(* PLC project Unnamed, Unknown Unnamed 1 *)
(* stored: creationDateTime 2012-09-12T23:30:19, modificationDateTime 2026-03-14T22:28:08 *)

FUNCTION_BLOCK getpybool
  VAR
    getpy : python_gear;
    latch : SR;
  END_VAR
  VAR_INPUT
    name : STRING;
  END_VAR
  VAR_OUTPUT
    val : BOOL;
  END_VAR
  VAR  (* added by the conversion: wires and edge detectors of the diagram *)
    _EQ41_ENO : BOOL;
    _EQ41_OUT : BOOL;
    _EQ3_ENO : BOOL;
    _EQ3_OUT : BOOL;
  END_VAR

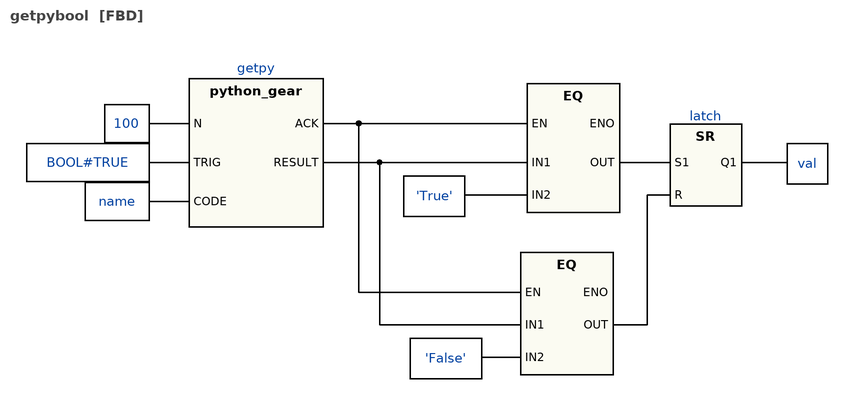
(* FBD diagram, written out as Structured Text *)
getpy(N := 100, TRIG := BOOL#TRUE, CODE := name);
_EQ41_OUT := EQ(EN := getpy.ACK, IN1 := getpy.RESULT, IN2 := 'True', ENO => _EQ41_ENO);
_EQ3_OUT := EQ(EN := getpy.ACK, IN1 := getpy.RESULT, IN2 := 'False', ENO => _EQ3_ENO);
latch(S1 := _EQ41_OUT, R := _EQ3_OUT);
val := latch.Q1;
END_FUNCTION_BLOCK

PROGRAM main
  VAR
    Done : BOOL;
  END_VAR
  VAR
    SlaveX AT %IW1.0.3.0 : AXIS_REF;
  END_VAR
  VAR
    SlaveY : AXIS_REF;
  END_VAR
  VAR
    Master AT %IW1.0.4.0 : AXIS_REF;
  END_VAR
  VAR
    switch : MC_Power;
    readpos : MC_ReadActualPosition;
    XPn : LREAL;
    YPn : LREAL;
    mPn : LREAL;
    XSetPoint : LREAL;
    XActualPos : LREAL;
    YVn : LREAL;
    mVn : LREAL;
    setpos : MC_SetPosition;
    readspeed : MC_ReadParameter;
    bt1 : getpybool;
    Block1 : getpybool;
    MC_Power0 : MC_Power;
    MC_ReadActualPosition0 : MC_ReadActualPosition;
    MC_SetPosition0 : MC_SetPosition;
    MC_ReadParameter0 : MC_ReadParameter;
    MC_MoveAbsolute0 : MC_MoveAbsolute;
    MC_CAM_REF_FROM_CSV0 : MC_CAM_REF_FROM_CSV;
    MC_CamTableSelect0 : MC_CamTableSelect;
    MC_CamIn0 : MC_CamIn;
    MC_CamOut0 : MC_CamOut;
    python_poll0 : python_gear;
    MC_CamTableSelect1 : MC_CamTableSelect;
    MC_CamIn1 : MC_CamIn;
    MC_CamOut1 : MC_CamOut;
    MC_Power1 : MC_Power;
    MC_ReadActualPosition1 : MC_ReadActualPosition;
    MC_SetPosition1 : MC_SetPosition;
    MC_ReadParameter1 : MC_ReadParameter;
    MC_Halt0 : MC_Halt;
    MC_ReadParameter2 : MC_ReadParameter;
    MC_Sim0 : MC_Sim;
    getpybool0 : getpybool;
  END_VAR
  VAR  (* added by the conversion: wires and edge detectors of the diagram *)
    F_TRIG1 : F_TRIG;
    F_TRIG2 : F_TRIG;
    F_TRIG3 : F_TRIG;
  END_VAR

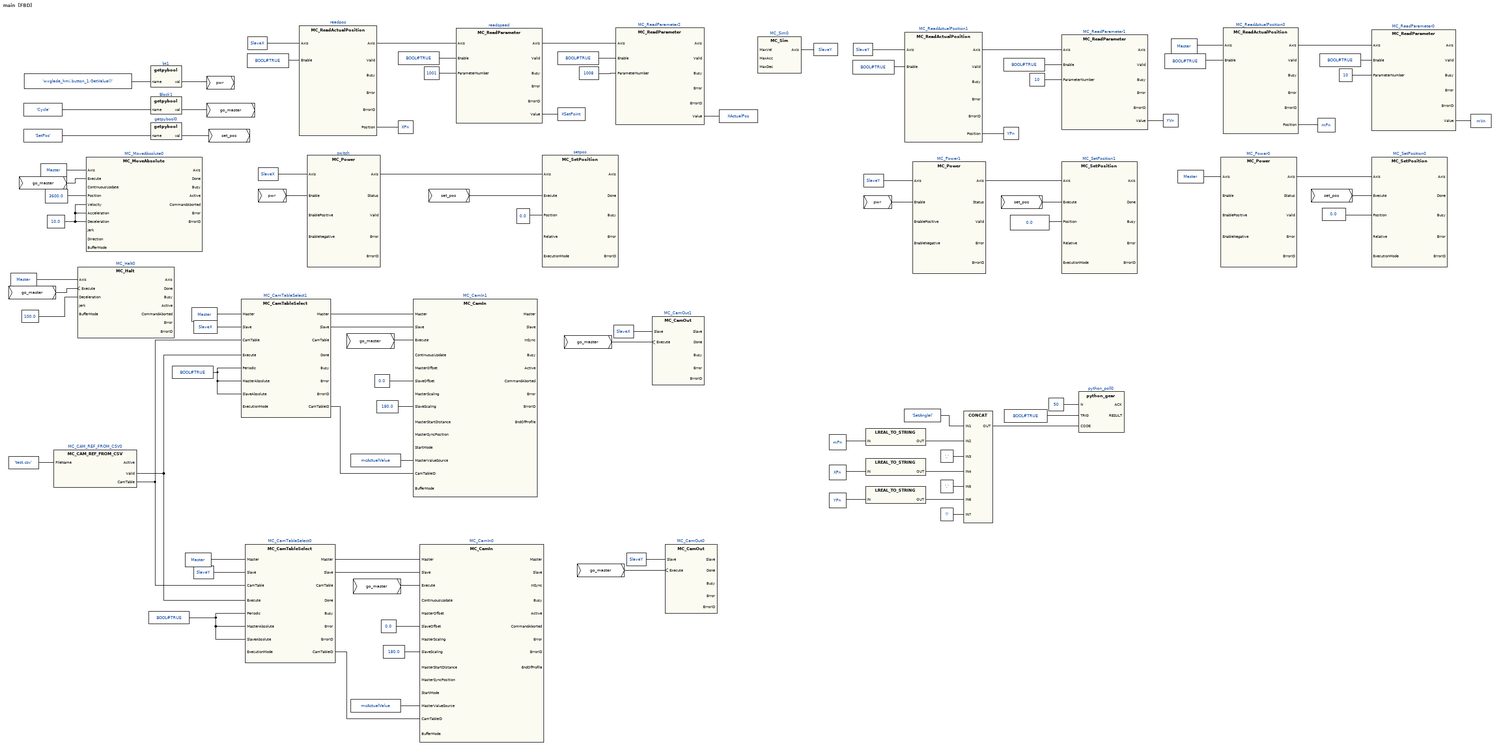
(* FBD diagram, written out as Structured Text *)
readpos(Axis := SlaveX, Enable := BOOL#TRUE);
XPn := readpos.Position;
readspeed(Axis := readpos.Axis, Enable := BOOL#TRUE, ParameterNumber := 1001);
XSetPoint := readspeed.Value;
MC_ReadActualPosition0(Axis := Master, Enable := BOOL#TRUE);
mPn := MC_ReadActualPosition0.Position;
MC_ReadParameter0(Axis := MC_ReadActualPosition0.Axis, Enable := BOOL#TRUE, ParameterNumber := 10);
mVn := MC_ReadParameter0.Value;
MC_ReadActualPosition1(Axis := SlaveY, Enable := BOOL#TRUE);
YPn := MC_ReadActualPosition1.Position;
MC_ReadParameter1(Axis := MC_ReadActualPosition1.Axis, Enable := BOOL#TRUE, ParameterNumber := 10);
YVn := MC_ReadParameter1.Value;
MC_ReadParameter2(Axis := readspeed.Axis, Enable := BOOL#TRUE, ParameterNumber := 1008);
XActualPos := MC_ReadParameter2.Value;
MC_Sim0();
SlaveY := MC_Sim0.Axis;
bt1(name := 'wxglade_hmi.button_1.GetValue()');
switch(Axis := SlaveX, Enable := bt1.val);
getpybool0(name := 'SetPos');
setpos(Axis := switch.Axis, Execute := getpybool0.val, Position := 0.0);
Block1(name := 'Cycle');
MC_Power0(Axis := Master);
MC_SetPosition0(Axis := MC_Power0.Axis, Execute := getpybool0.val, Position := 0.0);
MC_MoveAbsolute0(Axis := Master, Execute := Block1.val, Position := 3600.0, Velocity := 10.0, Acceleration := 10.0, Deceleration := 10.0);
MC_CAM_REF_FROM_CSV0(FileName := 'test.csv');
MC_CamTableSelect0(Master := Master, Slave := SlaveY, CamTable := MC_CAM_REF_FROM_CSV0.CamTable, Execute := MC_CAM_REF_FROM_CSV0.Valid, Periodic := BOOL#TRUE, MasterAbsolute := BOOL#TRUE, SlaveAbsolute := BOOL#TRUE);
MC_CamIn0(Master := MC_CamTableSelect0.Master, Slave := MC_CamTableSelect0.Slave, Execute := Block1.val, SlaveOffset := 0.0, SlaveScaling := 180.0, MasterValueSource := mcActualValue, CamTableID := MC_CamTableSelect0.CamTableID);
F_TRIG1(CLK := Block1.val);
MC_CamOut0(Slave := SlaveY, Execute := F_TRIG1.Q);
python_poll0(N := 50, TRIG := BOOL#TRUE, CODE := CONCAT('SetAngle(', LREAL_TO_STRING(mPn), ',', LREAL_TO_STRING(XPn), ',', LREAL_TO_STRING(YPn), ')'));
MC_CamTableSelect1(Master := Master, Slave := SlaveX, CamTable := MC_CAM_REF_FROM_CSV0.CamTable, Execute := MC_CAM_REF_FROM_CSV0.Valid, Periodic := BOOL#TRUE, MasterAbsolute := BOOL#TRUE, SlaveAbsolute := BOOL#TRUE);
MC_CamIn1(Master := MC_CamTableSelect1.Master, Slave := MC_CamTableSelect1.Slave, Execute := Block1.val, SlaveOffset := 0.0, SlaveScaling := 180.0, MasterValueSource := mcActualValue, CamTableID := MC_CamTableSelect1.CamTableID);
F_TRIG2(CLK := Block1.val);
MC_CamOut1(Slave := SlaveX, Execute := F_TRIG2.Q);
MC_Power1(Axis := SlaveY, Enable := bt1.val);
MC_SetPosition1(Axis := MC_Power1.Axis, Execute := getpybool0.val, Position := 0.0);
F_TRIG3(CLK := Block1.val);
MC_Halt0(Axis := Master, Execute := F_TRIG3.Q, Deceleration := 100.0);
END_PROGRAM

CONFIGURATION config
  RESOURCE resource1 ON PLC
    TASK tsk1(INTERVAL := T#1MS, PRIORITY := 0);
    PROGRAM inst1 WITH tsk1 : main;
  END_RESOURCE
END_CONFIGURATION
